// TIA Portal V19 export
DATA_BLOCK "RTrk"   // DB5
// stored: MemoryReserve 100
   VAR
      Last_RTrk_ID : DInt;   // Ultimo ID asseggnato a una foro di riferimento parte (Part/Semi-guscio)
   END_VAR
BEGIN
END_DATA_BLOCK
